// TIA Portal V20 export
FUNCTION "Block_2" : Void   // FC2, FBD
{ S7_Optimized_Access := 'TRUE' }
// stored: SetENOAutomatically false
BEGIN
END_FUNCTION
